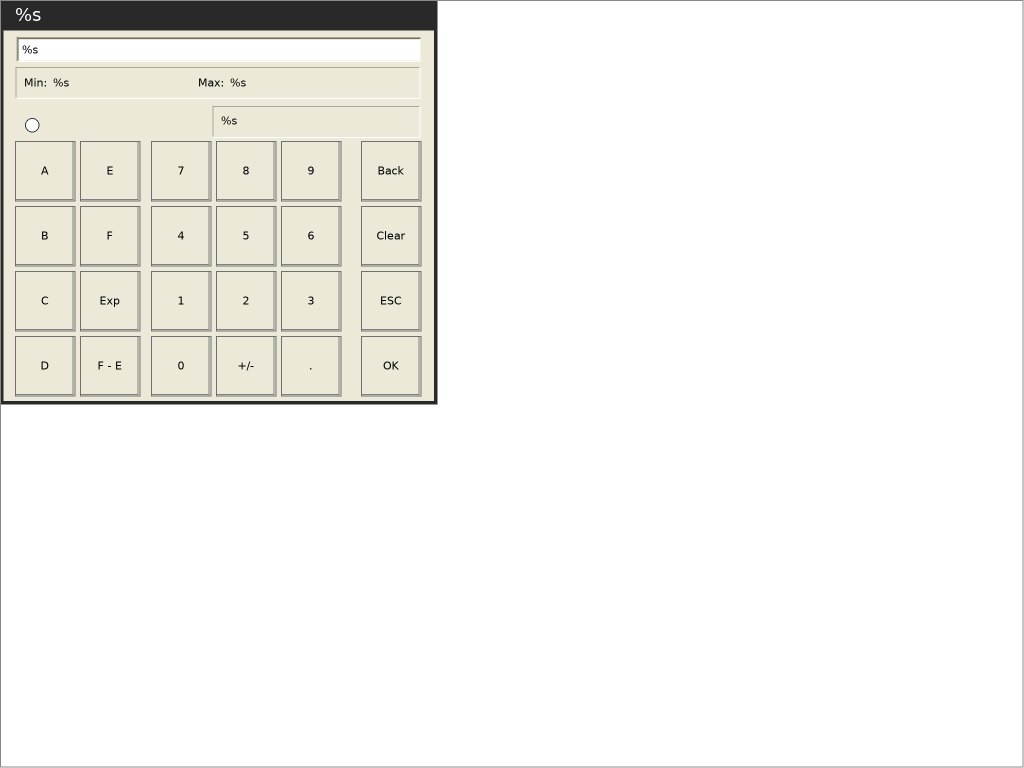
VISUALIZATION NumpadExtended  // 1024x768
VAR_INPUT
	stVariableValue : STRING;
	stMin : STRING;
	stMax : STRING;
	wstTitle : WSTRING;
	flags : DWORD;	
END_VAR
VAR
	bInit : BOOL;
	stMessage : STRING;
	// the display value
	stOutputValue : STRING;		
	// 0: dec, 1: hex, like Dialog_FormatTypes
	iFormatValue : INT;
	bInitFormatValue : BOOL;	
	iCaretPosition	: INT;
	iSelectionStart	: INT;
	iSelectionEnd	: INT;
	xAllSelected	: BOOL;
END_VAR
    Rectangle (3,29 434x39)
    Polyline (17,61) (17,37) (420,37)
    Polyline (18,61) (420,61) (420,38)
    Polyline (18,60) (18,38) (420,38)
    Textfield (19,40 400x20), "%s", text variable: stOutputValue
        p905179711: iCaretPosition
        p3815007873: iSelectionStart
        p1425650380: iSelectionEnd
        p3479897389: xAllSelected
    Rectangle (3,136 434x266)
    Button (361,336 60x60), "OK"
        OnMouseDown: execute { VisuDlgUtil_CloseNumpadExtended2(stOutputValue, stVariableValue, stMin, stMax, iFormatValue, bInitFormatValue, iCaretPosition, iSelectionStart, iSelectionEnd, flags); }
        OnMouseDown: CloseDialog Dialog=NumpadExtended, Result=OK, NumpadKeypad=True, NumpadKeypadSet=True
    Button (361,271 60x60), "ESC"
        OnMouseDown: execute { VisuDlgUtil_SetbInitFormatValue(bInitFormatValue, '0'); }
        OnMouseDown: CloseDialog Dialog=NumpadExtended, Result=Cancel, NumpadKeypad=True, NumpadKeypadSet=True
    Button (361,206 60x60), "Clear"
        OnMouseDown: execute { VisuDlg_ProcessClear(stOutputValue, stVariableValue, flags, iCaretPosition, iSelectionStart, iSelectionEnd); }
    Button (361,141 60x60), "Back"
        OnMouseDown: execute { VisuDlg_ProcessBack(stOutputValue, stVariableValue, iCaretPosition, iSelectionStart, iSelectionEnd, bInit); }
    Button (281,336 60x60), ".", input disabled if: iFormatValue = 1
        OnMouseDown: execute { VisuDlg_ProcessCharWithInit(stOutputValue, stVariableValue, iCaretPosition, iSelectionStart, iSelectionEnd, bInit, (flags AND VisuElems.Visu_InputFlags.Password) = 1, '.'); }
    Button (216,336 60x60), "+/-"
        OnMouseDown: execute { VisuDlg_ProcessChangeSignExtended(stOutputValue, stVariableValue, iCaretPosition, iSelectionStart, iSelectionEnd, bInit, (flags AND VisuElems.Visu_InputFlags.Password) = 1, iFormatValue); }
    Button (151,336 60x60), "0"
        OnMouseDown: execute { VisuDlg_ProcessCharWithInit(stOutputValue, stVariableValue, iCaretPosition, iSelectionStart, iSelectionEnd, bInit, (flags AND VisuElems.Visu_InputFlags.Password) = 1, '0'); }
    Button (151,271 60x60), "1"
        OnMouseDown: execute { VisuDlg_ProcessCharWithInit(stOutputValue, stVariableValue, iCaretPosition, iSelectionStart, iSelectionEnd, bInit, (flags AND VisuElems.Visu_InputFlags.Password) = 1, '1'); }
    Button (216,271 60x60), "2"
        OnMouseDown: execute { VisuDlg_ProcessCharWithInit(stOutputValue, stVariableValue, iCaretPosition, iSelectionStart, iSelectionEnd, bInit, (flags AND VisuElems.Visu_InputFlags.Password) = 1, '2'); }
    Button (281,271 60x60), "3"
        OnMouseDown: execute { VisuDlg_ProcessCharWithInit(stOutputValue, stVariableValue, iCaretPosition, iSelectionStart, iSelectionEnd, bInit, (flags AND VisuElems.Visu_InputFlags.Password) = 1, '3'); }
    Button (151,206 60x60), "4"
        OnMouseDown: execute { VisuDlg_ProcessCharWithInit(stOutputValue, stVariableValue, iCaretPosition, iSelectionStart, iSelectionEnd, bInit, (flags AND VisuElems.Visu_InputFlags.Password) = 1, '4'); }
    Button (216,206 60x60), "5"
        OnMouseDown: execute { VisuDlg_ProcessCharWithInit(stOutputValue, stVariableValue, iCaretPosition, iSelectionStart, iSelectionEnd, bInit, (flags AND VisuElems.Visu_InputFlags.Password) = 1, '5'); }
    Button (281,206 60x60), "6"
        OnMouseDown: execute { VisuDlg_ProcessCharWithInit(stOutputValue, stVariableValue, iCaretPosition, iSelectionStart, iSelectionEnd, bInit, (flags AND VisuElems.Visu_InputFlags.Password) = 1, '6'); }
    Button (151,141 60x60), "7"
        OnMouseDown: execute { VisuDlg_ProcessCharWithInit(stOutputValue, stVariableValue, iCaretPosition, iSelectionStart, iSelectionEnd, bInit, (flags AND VisuElems.Visu_InputFlags.Password) = 1, '7'); }
    Button (216,141 60x60), "8"
        OnMouseDown: execute { VisuDlg_ProcessCharWithInit(stOutputValue, stVariableValue, iCaretPosition, iSelectionStart, iSelectionEnd, bInit, (flags AND VisuElems.Visu_InputFlags.Password) = 1, '8'); }
    Button (281,141 60x60), "9"
        OnMouseDown: execute { VisuDlg_ProcessCharWithInit(stOutputValue, stVariableValue, iCaretPosition, iSelectionStart, iSelectionEnd, bInit, (flags AND VisuElems.Visu_InputFlags.Password) = 1, '9'); }
    Rectangle (3,67 434x69)
        p3560616238: VisuDlgUtil_InitValueFromFlags(flags, bInitFormatValue, iFormatValue)
    Rectangle (50,73 120x20), "%s", text variable: stMin, invisible if: LEN(stMin) = 0
    Rectangle (227,73 120x20), "%s", text variable: stMax, invisible if: LEN(stMax) = 0
    Rectangle (195,73 31x20), "Max:", text variable: stMin, invisible if: LEN(stMax) = 0
        p55702900: SEL(((UDINT_TO_DINT(flags AND 16#0010))=16#0010),16#FF000000,16#FFFF0000)
    Rectangle (296,401 3x3)
    Rectangle (434,0 3x404)
    Rectangle (0,0 3x404)
    Image (2,0 434x30), image: Title
    Rectangle (2,0 434x30), invisible if: VisuElems.g_VisualizationStyle.GetDINT('Dialog-UseHeaderColor', 0, 0) = 0
    Rectangle (12,5 406x20), "%s", text variable: wstTitle
    Rectangle (1,401 434x3)
    Polyline (213,136) (213,106) (419,106)
    Polyline (16,97) (16,67) (420,67)
    Polyline (213,137) (420,137) (420,106)
    Polyline (17,98) (420,98) (420,67)
    Rectangle (218,111 195x20), "%s", text variable: stMessage
    Rectangle (21,73 31x20), "Min:", text variable: stMin, invisible if: LEN(stMin) = 0
        p55702900: SEL(((UDINT_TO_DINT(flags AND 16#0008))=16#0008),16#FF000000,16#FFFF0000)
    Button (80,336 60x60), "F - E", input disabled if: iFormatValue = 1
        OnMouseDown: execute { VisuDlg_ProcessExpFloatFormatSwitch(stOutputValue, stVariableValue, iCaretPosition, iSelectionStart, iSelectionEnd, bInit, (flags AND VisuElems.Visu_InputFlags.Password) = 1); }
    Button (80,271 60x60), "Exp", input disabled if: iFormatValue = 1
        OnMouseDown: execute { VisuDlg_ProcessExp(stOutputValue, stVariableValue, iCaretPosition, iSelectionStart, iSelectionEnd, bInit, (flags AND VisuElems.Visu_InputFlags.Password) = 1); }
    Button (80,141 60x60), "E", input disabled if: iFormatValue = 0
        OnMouseDown: execute { VisuDlg_ProcessCharWithInit(stOutputValue, stVariableValue, iCaretPosition, iSelectionStart, iSelectionEnd, bInit, (flags AND VisuElems.Visu_InputFlags.Password) = 1, 'E'); }
    Button (80,206 60x60), "F", input disabled if: iFormatValue = 0
        OnMouseDown: execute { VisuDlg_ProcessCharWithInit(stOutputValue, stVariableValue, iCaretPosition, iSelectionStart, iSelectionEnd, bInit, (flags AND VisuElems.Visu_InputFlags.Password) = 1, 'F'); }
    Button (15,336 60x60), "D", input disabled if: iFormatValue = 0
        OnMouseDown: execute { VisuDlg_ProcessCharWithInit(stOutputValue, stVariableValue, iCaretPosition, iSelectionStart, iSelectionEnd, bInit, (flags AND VisuElems.Visu_InputFlags.Password) = 1, 'D'); }
    Button (15,271 60x60), "C", input disabled if: iFormatValue = 0
        OnMouseDown: execute { VisuDlg_ProcessCharWithInit(stOutputValue, stVariableValue, iCaretPosition, iSelectionStart, iSelectionEnd, bInit, (flags AND VisuElems.Visu_InputFlags.Password) = 1, 'C'); }
    Button (15,206 60x60), "B", input disabled if: iFormatValue = 0
        OnMouseDown: execute { VisuDlg_ProcessCharWithInit(stOutputValue, stVariableValue, iCaretPosition, iSelectionStart, iSelectionEnd, bInit, (flags AND VisuElems.Visu_InputFlags.Password) = 1, 'B'); }
    Button (15,141 60x60), "A", input disabled if: iFormatValue = 0
        OnMouseDown: execute { VisuDlg_ProcessCharWithInit(stOutputValue, stVariableValue, iCaretPosition, iSelectionStart, iSelectionEnd, bInit, (flags AND VisuElems.Visu_InputFlags.Password) = 1, 'A'); }
    RadioButton (23,110 150x30), variable: iFormatValue
        Areas[0]: Text=Dec
        Areas[1]: Text=Hex
    InvisibleInput (21,104 72x30)
        OnMouseDown: execute { VisuDlg_ProcessChangeNumberFormat(stOutputValue, stVariableValue, stMin, stMax, iFormatValue, iCaretPosition, iSelectionStart, iSelectionEnd, (flags AND VisuElems.Visu_InputFlags.Password) = 1, '0'); }
    InvisibleInput (96,104 72x30)
        OnMouseDown: execute { VisuDlg_ProcessChangeNumberFormat(stOutputValue, stVariableValue, stMin, stMax, iFormatValue, iCaretPosition, iSelectionStart, iSelectionEnd, (flags AND VisuElems.Visu_InputFlags.Password) = 1, '1'); }
END_VISUALIZATION

(* stored: Version 1.1.0.1, ProductVersion 3.1.4024.2
   Visu NumpadExtended: Id {c70b077b-7ed7-4e30-8b41-6461c7b1005c} *)
